TYPE
    SandboxData EXTENDS TcoData.TcoEntity :
    STRUCT
        sampleData : SampleDataStructure;
    END_STRUCT
END_TYPE

(* stored: Version 1.1.0.1, ProductVersion 3.1.4024.9
   DUT SandboxData: Id {db6560ed-fb2a-0049-1f52-f29952b65ec0} *)
